(*
Bufferd mode that is accumulated and bulk insert. Accumulated data size is calculated automatically among mininum/maximum_chunk_size parameter.
*)

FUNCTION_BLOCK BufferedRecord IMPLEMENTS IRecordDataQueue
VAR
	_current_index	: UDINT; // current index value
	_next_index 		: UDINT;
	sMeasurementName			: Tc2_System.T_MaxString;	// Measurement name of InfluxDB
	sSchemaName					: Tc2_System.T_MaxString;	// Schema name as a inserted data variable type name as structure
	min_chunk_size				: UDINT := DBLibParam.DATA_BUFFER_SIZE / 20;		// Minimum chunk size
	max_chunk_size				: UDINT	:= DBLibParam.DATA_BUFFER_SIZE;				// Maximum chunk size
	nDataBufferMaxIndex			: UDINT := DBLibParam.DATA_BUFFER_SIZE - 1;			// upper bound of data buffer array.
	_buffer_pointer : PVOID := 0;
	
	// Start point time
	start_time		: ULINT;
	start_data 		: T_Arg;

	nCycleTime		: UDINT;					// PLC task cycle time setting(in 100ns)
	data_size		: UDINT := 1;				// record data size
	accumulated_amount		: UDINT := 0;		// buffer usage
	last_data_count	: UDINT := 0;
	
	start_index		: UDINT;
	_buffer_usage	: REAL;				// data usage percentage of data buffer.
	_avalable_buffer_size	:DINT;
	diff_target		: REAL;
	pid_ope			: REAL;	
	chunk_size 		: UDINT;
	_recorder 		:IRecordDB;
	
END_VAR

(*Number of array items for data buffer*)
PROPERTY buffer_size : UDINT
GET
buffer_size := nDataBufferMaxIndex + 1;
END_GET
SET
IF buffer_size > 0 THEN
	nDataBufferMaxIndex := buffer_size - 1;	
END_IF
END_SET
END_PROPERTY

(* Usage of data buffer (0 - 1.0) [1/100%] *)
PROPERTY PUBLIC buffer_usage : REAL
GET
buffer_usage := _buffer_usage;
END_GET
END_PROPERTY

(* Structure name for each data model *)
PROPERTY PUBLIC data_def_structure_name : Tc2_System.T_MaxString
GET
END_GET
SET
sSchemaName := data_def_structure_name;
END_SET
END_PROPERTY

(* Database table(or measurement) name to which the data is inserted. *)
PROPERTY PUBLIC db_table_name : Tc2_System.T_MaxString
GET
END_GET
SET
sMeasurementName := db_table_name;
END_SET
END_PROPERTY

METHOD FB_init : BOOL
VAR_INPUT
	bInitRetains : BOOL; // if TRUE, the retain variables are initialized (warm start / cold start)
	bInCopyCode : BOOL;  // if TRUE, the instance afterwards gets moved into the copy code (online change)
	buffer_pointer :PVOID; // The pointer to data buffer that represent array of structured variable for bulk insert. 
	recorder	:IRecordDB; // IRecordDB is a interface class of database connection endpoint object.
END_VAR
_buffer_pointer := buffer_pointer;
_recorder := recorder;
END_METHOD

(* Current index of data buffer array *)
PROPERTY index : UDINT
GET
index := _current_index;
END_GET
END_PROPERTY

PROPERTY PUBLIC maximum_chunk_size : UDINT
GET
maximum_chunk_size := max_chunk_size;
END_GET
SET
max_chunk_size := maximum_chunk_size;
END_SET
END_PROPERTY

PROPERTY PUBLIC minimum_chunk_size : UDINT
GET
minimum_chunk_size := min_chunk_size;
END_GET
SET
min_chunk_size := minimum_chunk_size;
END_SET
END_PROPERTY

(* The target buffer index at which assume the data in buffer reaches specified size and bulk insert command be sent to database engine.  *)
PROPERTY next_index : UDINT
GET
next_index := _next_index;
END_GET
END_PROPERTY

(*The method to write to database through data buffer with queue.*)
{warning 'add method implementation '}
METHOD write : BOOL // Return true if data is put on buffer queue successfully.
VAR_INPUT
	input_data	: T_Arg;	// Set the measured data. It should be same data type as item of data buffer that is set at "buffer_pointer" on "FB_init" constructor.
END_VAR
VAR
	gCurrentData	:T_Arg;
	pCurrentBufferPointer : PVOID;
	work_data_body  :DbInsertCommand;
END_VAR
IF _recorder = 0 THEN
	write := FALSE;
	RETURN;
END_IF

pCurrentBufferPointer := _buffer_pointer + input_data.cbLen * _current_index;
MEMCPY(pCurrentBufferPointer, input_data.pData, input_data.cbLen);
gCurrentData := F_BIGTYPE(pData := pCurrentBufferPointer, cbLen := input_data.cbLen);

IF _current_index = start_index THEN
	start_time := F_GetSystemTime();
	start_data := gCurrentData;
END_IF

IF _next_index <= _current_index OR _current_index >= nDataBufferMaxIndex THEN
	max_chunk_size := nDataBufferMaxIndex + 1;
	// put_data
	IF NOT _recorder.queue.full THEN
		data_size := _current_index - start_index + 1;
		_avalable_buffer_size := UDINT_TO_DINT(nDataBufferMaxIndex) - UDINT_TO_DINT(accumulated_amount) +1;
		IF _avalable_buffer_size < UDINT_TO_DINT(data_size) AND _avalable_buffer_size > 0 THEN
			data_size := DINT_TO_UDINT(_avalable_buffer_size);
		ELSIF _avalable_buffer_size <= 0 THEN
			data_size := 0;
		END_IF

		IF data_size > 1 THEN
			
			// calculate each cycle time by num of data among start time and current time.
			nCycleTime := ULINT_TO_UDINT(F_GetSystemTime() - start_time) / (data_size - 1);
			work_data_body.data_body := start_data;
			work_data_body.start_time := start_time;
			work_data_body.cycle_time_100ns := nCycleTime;
			work_data_body.chunk_size := data_size;
			work_data_body.MeasurementName := sMeasurementName;
			work_data_body.SchemaName := sSchemaName;
			work_data_body.accumulated_amount REF= accumulated_amount;
			// queue in
			_recorder.queue.put(work_data_body);
			start_index := _current_index + 1;
		END_IF
	END_IF
END_IF


IF last_data_count <> accumulated_amount THEN
	// calculate next index
	_buffer_usage := UDINT_TO_REAL(accumulated_amount) / UDINT_TO_REAL(nDataBufferMaxIndex + 1);
	diff_target := UDINT_TO_REAL(max_chunk_size) * _buffer_usage;
	pid_ope := UDINT_TO_REAL(min_chunk_size) + diff_target;
	chunk_size := REAL_TO_UDINT(pid_ope);
	//chunk_size := minimum_chunk_size;
	_next_index := _current_index + chunk_size - 1;
	IF chunk_size < min_chunk_size OR pid_ope < 0 THEN
		chunk_size := min_chunk_size;
	ELSIF chunk_size > max_chunk_size THEN
		chunk_size := max_chunk_size;
	END_IF
END_IF

last_data_count := accumulated_amount;

IF _current_index < nDataBufferMaxIndex THEN
	_current_index := _current_index + 1;
ELSE
	_current_index := 0;
	start_index := 0;
	_next_index := chunk_size - 1;
END_IF

write := TRUE;
END_METHOD

END_FUNCTION_BLOCK

(* stored: Version 1.1.0.1, ProductVersion 3.1.4024.12
   POU BufferedRecord: Id {8b3999e3-c2e1-4344-9092-4e707723d89a}, SpecialFunc None
   Property buffer_size: Id {b36ce7a6-bd18-43aa-8301-c9010135cc3f}
   Get Get: Id {2b913049-e685-41f9-94f3-9003bf0289f3}
   Set Set: Id {ced6233f-4469-42d7-a5b7-58237174f40c}
   Property buffer_usage: Id {bbb95211-74e1-4da1-9e2b-be2248fb01e5}
   Get Get: Id {b46d5d51-f7df-45ba-9aab-0d3c72cb9324}
   Property data_def_structure_name: Id {12d15a2c-bf0d-4db7-a907-7cebd338c4d6}
   Get Get: Id {ebda072e-3d15-41ca-8ab8-cbbe755d7e35}
   Set Set: Id {374779eb-84af-449b-b1d1-d49d94a7b136}
   Property db_table_name: Id {457088bd-30e0-4a96-b934-15df6743d6b6}
   Get Get: Id {4d8d5759-a539-49cb-92e4-0c653a06c4e1}
   Set Set: Id {5583acd3-dff8-4ba3-acf1-2446e6b0a828}
   Method FB_init: Id {60fdb3e5-25f4-4374-8251-80149f28a778}
   Property index: Id {14045ef6-f59e-4a14-bab6-425c44445155}
   Get Get: Id {ffbd4f52-8e5e-4810-9b2a-1a43f99167d3}
   Property maximum_chunk_size: Id {02c2c686-c7db-499b-a50c-3e861736b577}
   Get Get: Id {0baff072-67eb-4a7c-8fad-76d523574483}
   Set Set: Id {59369926-4939-4df1-910f-88ccb0b731a6}
   Property minimum_chunk_size: Id {7194ace4-c543-4d3b-bb4c-7732e82ecf0f}
   Get Get: Id {a7346a3e-d6df-4d67-acd9-15108b0b7d1f}
   Set Set: Id {bf381183-3550-45b7-9d0d-d87b431cae4d}
   Property next_index: Id {f5a3ffd6-3bc9-426f-b681-aff2cae57f4f}
   Get Get: Id {6789c059-d92d-49d3-96f5-eb79ca9b5e2b}
   Method write: Id {4d6a4f57-2187-4032-b3a4-3e31e3263b61} *)
